DATA_BLOCK "IAI_A3"
{ S7_Optimized_Access := 'FALSE' }
VERSION : 0.1
NON_RETAIN
// ATTRIBUTES
// AUTO_NUMBER = False
// BLOCK_NUMBER = 2213
// END_ATTRIBUTES
   STRUCT
      In : Struct
         iInterlock : Bool;
         "iManJog+" : Bool;
         "iManJog-" : Bool;
         iAutoStart : Bool;
         iHome : Bool;
         iCancelTask : Bool;
         iPauseTask : Bool;
         iManStart : Bool;
         iManListStart : Bool;
         iLimitSwitchActive : Bool;
         iLimitSoftActive : Bool;
         iRunningTimeout : Time;
         iHomingTimeout : Time;
         iAutoPosition : DInt;
         iAutoVelocity : Int;
         iManListPosition : DInt;
         iManListVelocity : Int;
         iManListNumber : Int;
         iManPosition : DInt;
         iManVelocity : Int;
         iMode : Int;
      END_STRUCT;
      Out : Struct
         oReady : Bool;
         oWarning : Bool;
         oError : Bool;
         oInterlock : Bool;
         oServoEnable : Bool;
         oRunning : Bool;
         oHoming : Bool;
         oHomeRef : Bool;
         oServoPosOK : Bool;
         oErrorCode : Int;
         oStatus : Int;
         oActPosition : DInt;
         oManualListPos : DInt;
      END_STRUCT;
      IO : Struct
         ioManEnale : Bool;
         ioAutoEnale : Bool;
      END_STRUCT;
      Spare : Struct
         S : Array[0..100] of Byte;
      END_STRUCT;
      Manual : Struct
         Index : Int;
         Pos : Array[1..20] of Struct
            Pos : Real;
            Vel : Int;
         END_STRUCT;
      END_STRUCT;
      Auto : Struct
         Index : Int;
         Pos : Array[1..20] of Struct
            Pos : Real;
            Vel : Int;
         END_STRUCT;
      END_STRUCT;
      Interlock : Struct
         Active : Bool;
         Case1 : Bool;
         Case2 : Bool;
         Case3 : Bool;
         Case4 : Bool;
         Case5 : Bool;
         Case6 : Bool;
         Case7 : Bool;
         Case8 : Bool;
         Case9 : Bool;
         Case10 : Bool;
      END_STRUCT;
      PositionOk : Array[1..20] of Bool;
      Home_Pos : Struct
         "Home Pos Pls" : Bool;
         "Arrow indication" : Int;
         "Process prompt" : Int;
         "Button prompt" : Int;
      END_STRUCT;
   END_STRUCT;


BEGIN
   In.iLimitSwitchActive := true;
   In.iLimitSoftActive := true;
   Manual.Index := 1;
   Auto.Index := 1;

END_DATA_BLOCK

